// TIA Portal V17 export
// export: Created 2024-09-02T12:50:34.2462658Z, ExportSetting WithDefaults, DisplayName Totally Integrated Automation Portal, DisplayVersion V17, DisplayName TIA Portal Openness, DisplayVersion V17, DisplayName TIA Portal Version Control Interface, DisplayVersion V17, DisplayName STEP 7 Professional, DisplayVersion V17, DisplayName STEP 7 Safety, DisplayVersion V17, DisplayName WinCC Professional, DisplayVersion V17
TYPE "typ_MobyDatenQPress"
// stored: IsFailsafeCompliant false
   STRUCT
      Datenkennung_00 { ExternalWritable := 'False'} : Array[0..1] of Char;
      TAF_Nummer_02 { ExternalWritable := 'False'} : Array[0..3] of Char;
      Compac_Errors_06 { ExternalWritable := 'False'} : Byte;
      Compac_Errors_07 { ExternalWritable := 'False'} : Byte;
      Einpressstelle_08 { ExternalWritable := 'False'} : Array[0..3] of Char;
      Einpresskraft_Ist_12 { ExternalWritable := 'False'} : DInt;
      Einpresskraft_Min_16 { ExternalWritable := 'False'} : DInt;
      Einpresskraft_Max_20 { ExternalWritable := 'False'} : DInt;
      Weg_Ist_24 { ExternalWritable := 'False'} : Int;
      Weg_Min_26 { ExternalWritable := 'False'} : Int;
      Weg_Max_28 { ExternalWritable := 'False'} : Int;
   END_STRUCT;
END_TYPE
